PROGRAM MAIN
VAR
	
END_VAR

//main program
INIT();

//SUBMQTT Connection and receiving
//submqtt();

//FTP
FTP();

//AT COmmands decoder
//commandDecoder();

//Get positions
POSITION();

//Error
ERROR();

END_PROGRAM

(* stored: Version 1.1.0.1, ProductVersion 3.1.4022.17
   POU MAIN: Id {f3e90440-582f-45a4-ac51-5f2449296ba8}, SpecialFunc None *)
